Universal Robots PolyScope program: TEST_SUB_104RXFF.urp

Program TEST_SUB_104RXFF (installation=GD directory=/programs/GD createdIn=5.13.0 lastSavedIn=5.13.0 robotSerialNumber=20205000017)
Calibrated DH parameters: a=[-0.000157, -0.56303, -0.236706, -0.000074, -0.000109, 0]; d=[0.181705, 47.632387, 369.599619, -417.058513, 0.119878, 0.115667]; alpha=[1.570881, -0.005074, -0.001247, 1.56886, -1.570997, 0]; deltaTheta=[0, -0.405485, 5.544791, 1.143886, -0.000009, -0.000001]
InitVariablesNode
BeforeStart
  Script file /programs/GD/CONTROL/FORCE_CONTROL.script
    | def GET_TCP_FORCE_TOOL():
    |   force_torque=get_tcp_force()
    |   force_B=p[force_torque[0], force_torque[1], force_torque[2], 0, 0, 0]
    |   torque_B=p[force_torque[3], force_torque[4], force_torque[5], 0, 0, 0]
    |   tcp=get_actual_tcp_pose()
    |   rotation_BT=p[0, 0, 0, tcp[3], tcp[4], tcp[5]]
    |   force_T=pose_trans(pose_inv(rotation_BT), force_B)
    |   torque_T=pose_trans(pose_inv(rotation_BT), torque_B)
    |   force_torque_T=p[force_T[0], force_T[1], force_T[2], torque_T[0], torque_T[1], torque_T[2]]
    |   return force_torque_T
    | end
Robot Program (runOnlyOnce=true)
  SuppressedNode
    Script: SET_BUCKET()
  SuppressedNode
    Folder ROVI_CAPTURE
      If ( not ROVI_CAPTURE())
        SubPrgResult := rovi_err
        Wait Sleep waitTime=999999
      CandCnt := Y1[0]
      DistPillar := Y1[1] / 1000.0
      LevelZ := Y1[2] / 1000.0
      NeighborZ := Y1[3] / 1000.0
      If (GP_int_in[0]==1201)
        DistPillarBak := DistPillar
      If (CandCnt<1)
        SubPrgResult := 990
        Wait Sleep waitTime=999999
  SuppressedNode
    Folder ROVI_SOLVE
      If (CandCnt>0)
        Y2 := ROVI_SOLVE()
        If (Y2[0]≟10000.)
          SubPrgResult := rovi_err
          Wait Sleep waitTime=999999
  SuppressedNode
    UF := Y2
  DistPillar := 0.5
  Folder PICK
    SetPayload (workpieceName=k10)
    '1=MOVE'
    '2=MOVE+FIXEDBALANCE'
    '3=FORCEMOVE'
    '4=FORCEZ'
    '5=FORCEZ+WEAVE'
    '6=[LM]FORCEZ+WEAVE'
    '7=[RM]FORCEZ+WEAVE'
    '8=[RM]FORCEZ'
    i := 8
    Loop Counting (count=3) loopVariable(name=ループ_1)
      Switch expression=i
        Case (caseValue=1)
          MoveL speed 400 mm/s, acceleration 70 mm/s^2 (useActiveTCP=false) tcp=TCP_RX; feature=UF
            Waypoint Variable (Variable): variable(featureName=gGD_3_M_RX)
            Waypoint Variable (Variable): variable(featureName=gGD_2_M_RX)
            Wait Sleep waitTime=0.5
            SuppressedNode
              Popup Message (haltProgram=false message=ok? inputType=Text)
            Waypoint Variable (Variable): variable(featureName=gGD_1_M_RX)
        Case (caseValue=2)
          MoveL speed 400 mm/s, acceleration 70 mm/s^2 (useActiveTCP=false) tcp=TCP_RX; feature=UF
            Waypoint Variable (Variable): variable(featureName=gGD_3_M_RX)
            Waypoint Variable (Variable): variable(featureName=gGD_2_M_RX)
            Set SingleDigitalPulseActionState SingleDigitalPulseActionState(hiPulseInSeconds=1, pin=GP_bool_out[14])
            Wait Sleep waitTime=0.5
            SuppressedNode
              Popup Message (haltProgram=false message=ok? inputType=Text)
            Waypoint Variable (Variable): variable(featureName=gGD_1_M_RX)
            Set SingleDigitalPulseActionState SingleDigitalPulseActionState(hiPulseInSeconds=1, pin=GP_bool_out[15])
        Case (caseValue=3)
          MoveL speed 400 mm/s, acceleration 70 mm/s^2 (useActiveTCP=false) tcp=TCP_RX; feature=UF
            Waypoint Variable (Variable): variable(featureName=gGD_3_M_RX)
            Waypoint Variable (Variable): variable(featureName=gGD_2_M_RX)
            Set SingleDigitalPulseActionState SingleDigitalPulseActionState(hiPulseInSeconds=1, pin=GP_bool_out[14])
            Wait Sleep waitTime=0.5
            SuppressedNode
              Popup Message (haltProgram=false message=ok? inputType=Text)
          Force Frame feature=Joint_6_name; selection=[1, 1, 0, 0, 0, 0]; wrench=[0, 0, 0, 0, 0, 0]; limitsForce=[0.005, 0.005, 0.03, 1.047198, 1.047198, 1.047198]; limitsMotion=[0.1, 0.1, 0.1, 0.349066, 0.349066, 0.349066]
            MoveL speed 120 mm/s, acceleration 70 mm/s^2 (useActiveTCP=false) tcp=TCP_RX; feature=UF
              Waypoint Variable (Variable): variable(featureName=gGD_1_M_RX)
          Set SingleDigitalPulseActionState SingleDigitalPulseActionState(hiPulseInSeconds=1, pin=GP_bool_out[15])
        Case (caseValue=4)
          MoveL speed 400 mm/s, acceleration 70 mm/s^2 (useActiveTCP=false) tcp=TCP_RX; feature=UF
            Waypoint Variable (Variable): variable(featureName=gGD_3_M_RX)
            Waypoint Variable (Variable): variable(featureName=gGD_2_M_RX)
            Set SingleDigitalPulseActionState SingleDigitalPulseActionState(hiPulseInSeconds=1, pin=GP_bool_out[14])
            Wait Sleep waitTime=0.5
            SuppressedNode
              Popup Message (haltProgram=false message=ok? inputType=Text)
          Force Frame feature=Joint_6_name; selection=[1, 1, 1, 0, 0, 0]; wrench=[0, 0, 10, 0, 0, 0]; limitsForce=[0.005, 0.005, 0.03, 0.034907, 0.034907, 1.047198]; limitsMotion=[0.1, 0.1, 0.1, 0.349066, 0.349066, 0.349066]
            Wait Condition expression=CurrPos_p[1]≤(gGD_1_M_RX[1]-0.015)
          Popup Message (haltProgram=false message=ok inputType=Text)
          Set SingleDigitalPulseActionState SingleDigitalPulseActionState(hiPulseInSeconds=1, pin=GP_bool_out[15])
        Case (caseValue=5)
          MoveL speed 400 mm/s, acceleration 70 mm/s^2 (useActiveTCP=false) tcp=TCP_RX; feature=UF
            Waypoint Variable (Variable): variable(featureName=gGD_3_M_RX)
            Waypoint Variable (Variable): variable(featureName=gGD_2_M_RX)
            Set SingleDigitalPulseActionState SingleDigitalPulseActionState(hiPulseInSeconds=1, pin=GP_bool_out[14])
            Wait Sleep waitTime=0.5
            SuppressedNode
              Popup Message (haltProgram=false message=ok? inputType=Text)
          Sub3100_Option := 9
          Force Frame feature=Joint_6_name; selection=[1, 1, 1, 0, 0, 0]; wrench=[0, 0, 10, 0, 0, 0]; limitsForce=[0.005, 0.005, 0.03, 0.034907, 0.034907, 1.047198]; limitsMotion=[0.1, 0.1, 0.1, 0.349066, 0.349066, 0.349066]
            Loop While (checkContinuously=false) expression=CurrPos_p[1]>(gGD_1_M_RX[1]-0.015)
              If tcp_speed[2]<0.0005
                '7:RX+,8:RX-,9:RY+,10:RY-,11:RZ+,12:RZ-'
                Sub3100_Xd := [0.,0.,0.,0.,0.,0.]
                Sub3100_q := floor((Sub3100_Option-1) / 2)
                Sub3100_e := 1-((Sub3100_Option-1) % 2)*2
                Sub3100_t := 0.2
                Script: Sub3100_Xd[Sub3100_q]=d2r(Sub3100_XdRot)*Sub3100_e
                Script: speedl(Sub3100_Xd,Sub3100_aRot,Sub3100_t)
                If Sub3100_Option≟9
                  Sub3100_Option := 10
                Else 
                  Sub3100_Option := 9
          Popup Message (haltProgram=false message=ok inputType=Text)
          Set SingleDigitalPulseActionState SingleDigitalPulseActionState(hiPulseInSeconds=1, pin=GP_bool_out[15])
        Case (caseValue=6)
          MoveL speed 400 mm/s, acceleration 70 mm/s^2 (useActiveTCP=false) tcp=TCP_RX; feature=UF
            Waypoint Variable (Variable): variable(featureName=gGD_3_LM_RX)
            Waypoint Variable (Variable): variable(featureName=gGD_2_LM_RX)
            Set SingleDigitalPulseActionState SingleDigitalPulseActionState(hiPulseInSeconds=1, pin=GP_bool_out[14])
            Wait Sleep waitTime=0.5
            SuppressedNode
              Popup Message (haltProgram=false message=ok? inputType=Text)
          Sub3100_Option := 9
          Force Frame feature=Joint_6_name; selection=[1, 1, 1, 0, 0, 0]; wrench=[0, 0, 10, 0, 0, 0]; limitsForce=[0.005, 0.005, 0.03, 0.034907, 0.034907, 1.047198]; limitsMotion=[0.1, 0.1, 0.1, 0.349066, 0.349066, 0.349066]
            Loop While (checkContinuously=false) expression=CurrPos_p[1]>(gGD_1_LM_RX[1]-0.015)
              If tcp_speed[2]<0.0005
                '7:RX+,8:RX-,9:RY+,10:RY-,11:RZ+,12:RZ-'
                Sub3100_Xd := [0.,0.,0.,0.,0.,0.]
                Sub3100_q := floor((Sub3100_Option-1) / 2)
                Sub3100_e := 1-((Sub3100_Option-1) % 2)*2
                Sub3100_t := 0.2
                Script: Sub3100_Xd[Sub3100_q]=d2r(Sub3100_XdRot)*Sub3100_e
                Script: speedl(Sub3100_Xd,Sub3100_aRot/2.0,Sub3100_t)
                If Sub3100_Option≟9
                  Sub3100_Option := 10
                Else 
                  Sub3100_Option := 9
          Popup Message (haltProgram=false message=ok inputType=Text)
          Set SingleDigitalPulseActionState SingleDigitalPulseActionState(hiPulseInSeconds=1, pin=GP_bool_out[15])
        Case (caseValue=7)
          MoveL speed 400 mm/s, acceleration 70 mm/s^2 (useActiveTCP=false) tcp=TCP_RX; feature=UF
            Waypoint Variable (Variable): variable(featureName=gGD_3_RM_RX)
            Waypoint Variable (Variable): variable(featureName=gGD_2_RM_RX)
            Set SingleDigitalPulseActionState SingleDigitalPulseActionState(hiPulseInSeconds=1, pin=GP_bool_out[14])
            Wait Sleep waitTime=0.5
            SuppressedNode
              Popup Message (haltProgram=false message=ok? inputType=Text)
          Sub3100_Option := 9
          Force Frame feature=Joint_6_name; selection=[1, 1, 1, 0, 0, 0]; wrench=[0, 0, 10, 0, 0, 0]; limitsForce=[0.005, 0.005, 0.03, 0.034907, 0.034907, 1.047198]; limitsMotion=[0.1, 0.1, 0.1, 0.349066, 0.349066, 0.349066]
            Loop While (checkContinuously=false) expression=CurrPos_p[1]>(gGD_1_RM_RX[1]-0.015)
              If tcp_speed[2]<0.0005
                '7:RX+,8:RX-,9:RY+,10:RY-,11:RZ+,12:RZ-'
                Sub3100_Xd := [0.,0.,0.,0.,0.,0.]
                Sub3100_q := floor((Sub3100_Option-1) / 2)
                Sub3100_e := 1-((Sub3100_Option-1) % 2)*2
                Sub3100_t := 0.2
                Script: Sub3100_Xd[Sub3100_q]=d2r(Sub3100_XdRot)*Sub3100_e
                Script: speedl(Sub3100_Xd,Sub3100_aRot/2.0,Sub3100_t)
                If Sub3100_Option≟9
                  Sub3100_Option := 10
                Else 
                  Sub3100_Option := 9
          Popup Message (haltProgram=false message=ok inputType=Text)
          Set SingleDigitalPulseActionState SingleDigitalPulseActionState(hiPulseInSeconds=1, pin=GP_bool_out[15])
        Case (caseValue=8)
          MoveL speed 400 mm/s, acceleration 70 mm/s^2 (useActiveTCP=false) tcp=TCP_RX; feature=UF
            Waypoint Variable (Variable): variable(featureName=gGD_3_RM_RX)
            Waypoint Variable (Variable): variable(featureName=gGD_2_RM_RX)
            Set SingleDigitalPulseActionState SingleDigitalPulseActionState(hiPulseInSeconds=1, pin=GP_bool_out[14])
            Wait Sleep waitTime=0.5
            SuppressedNode
              Popup Message (haltProgram=false message=ok? inputType=Text)
          Force Frame feature=Joint_6_name; selection=[1, 1, 1, 0, 0, 0]; wrench=[0, 0, 10, 0, 0, 0]; limitsForce=[0.005, 0.005, 0.03, 0.034907, 0.034907, 1.047198]; limitsMotion=[0.1, 0.1, 0.1, 0.349066, 0.349066, 0.349066]
            Wait Condition expression=CurrPos_p[1]≤(gGD_1_RM_RX[1]-0.015)
          Popup Message (haltProgram=false message=ok inputType=Text)
          Set SingleDigitalPulseActionState SingleDigitalPulseActionState(hiPulseInSeconds=1, pin=GP_bool_out[15])
      If i<6
        MoveL speed 400 mm/s, acceleration 70 mm/s^2 (useActiveTCP=false) tcp=TCP_RX; feature=UF
          Waypoint Variable (Variable): variable(featureName=gGD_2_M_RX)
          Waypoint Variable (Variable): variable(featureName=gGD_3_M_RX)
      ElseIf i≟6
        MoveL speed 400 mm/s, acceleration 70 mm/s^2 (useActiveTCP=false) tcp=TCP_RX; feature=UF
          Waypoint Variable (Variable): variable(featureName=gGD_2_LM_RX)
          Waypoint Variable (Variable): variable(featureName=gGD_3_LM_RX)
      Else 
        MoveL speed 400 mm/s, acceleration 70 mm/s^2 (useActiveTCP=false) tcp=TCP_RX; feature=UF
          Waypoint Variable (Variable): variable(featureName=gGD_2_RM_RX)
          Waypoint Variable (Variable): variable(featureName=gGD_3_RM_RX)
      Wait Sleep waitTime=4
    Halt
    If (0≤DistPillar and DistPillar≤DistPillarAPTh)
      MoveL speed 400 mm/s, acceleration 140 mm/s^2 (useActiveTCP=false) tcp=TCP_1; feature=UF
        Waypoint Variable (Variable): variable(featureName=gGD_4_LM)
      MoveL speed 400 mm/s, acceleration 140 mm/s^2 (useActiveTCP=false) tcp=TCP_RX; feature=UF
        Waypoint Variable (Variable): variable(featureName=gGD_3_LM_RX)
        Waypoint Variable (Variable): variable(featureName=gGD_2_LM_RX)
        Set SingleDigitalPulseActionState SingleDigitalPulseActionState(hiPulseInSeconds=1, pin=GP_bool_out[14])
        Wait Sleep waitTime=0.5
        SuppressedNode
          Popup Message (haltProgram=false message=ok? inputType=Text)
        Waypoint Variable (Variable): variable(featureName=gGD_1_LM_RX)
      Sub3100_Option := 9
      Force Frame feature=Joint_6_name; selection=[1, 1, 1, 0, 0, 0]; wrench=[0, 0, 10, 0, 0, 0]; limitsForce=[0.005, 0.005, 0.03, 0.034907, 0.034907, 1.047198]; limitsMotion=[0.1, 0.1, 0.1, 0.349066, 0.349066, 0.349066]
        Loop While (checkContinuously=false) expression=CurrPos_p[1]>(gGD_1_M_RX[1]-0.015)
          If tcp_speed[2]<0.0005
            '7:RX+,8:RX-,9:RY+,10:RY-,11:RZ+,12:RZ-'
            Sub3100_Xd := [0.,0.,0.,0.,0.,0.]
            Sub3100_q := floor((Sub3100_Option-1) / 2)
            Sub3100_e := 1-((Sub3100_Option-1) % 2)*2
            Sub3100_t := 0.2
            Script: Sub3100_Xd[Sub3100_q]=d2r(Sub3100_XdRot)*Sub3100_e
            Script: speedl(Sub3100_Xd,Sub3100_aRot,Sub3100_t)
            If Sub3100_Option≟9
              Sub3100_Option := 10
            Else 
              Sub3100_Option := 9
      Set SingleDigitalPulseActionState SingleDigitalPulseActionState(hiPulseInSeconds=1, pin=GP_bool_out[15])
    ElseIf (-DistPillarAPTh≤DistPillar and DistPillar≤0)
      MoveL speed 400 mm/s, acceleration 70 mm/s^2 (useActiveTCP=false) tcp=TCP_1; feature=UF
        Waypoint Variable (Variable): variable(featureName=gGD_4_RM)
      MoveL speed 400 mm/s, acceleration 70 mm/s^2 (useActiveTCP=false) tcp=TCP_RX; feature=UF
        Waypoint Variable (Variable): variable(featureName=gGD_3_RM_RX)
        Waypoint Variable (Variable): variable(featureName=gGD_2_RM_RX)
        Wait Sleep waitTime=0.5
        SuppressedNode
          Popup Message (haltProgram=false message=ok? inputType=Text)
        Waypoint Variable (Variable): variable(featureName=gGD_1_RM_RX)
    Else 
      MoveL speed 400 mm/s, acceleration 70 mm/s^2 (useActiveTCP=false) tcp=TCP_RX; feature=UF
        Waypoint Variable (Variable): variable(featureName=gGD_3_M_RX)
        Waypoint Variable (Variable): variable(featureName=gGD_2_M_RX)
        Set SingleDigitalPulseActionState SingleDigitalPulseActionState(hiPulseInSeconds=1, pin=GP_bool_out[14])
        Wait Sleep waitTime=0.5
        SuppressedNode
          Popup Message (haltProgram=false message=ok? inputType=Text)
      Force Frame feature=Joint_6_name; selection=[1, 1, 0, 0, 0, 0]; wrench=[0, 0, 0, 0, 0, 0]; limitsForce=[0.005, 0.005, 0.03, 1.047198, 1.047198, 1.047198]; limitsMotion=[0.1, 0.1, 0.1, 0.349066, 0.349066, 0.349066]
        MoveL speed 120 mm/s, acceleration 70 mm/s^2 (useActiveTCP=false) tcp=TCP_RX; feature=UF
          Waypoint Variable (Variable): variable(featureName=gGD_1_M_RX)
      Set SingleDigitalPulseActionState SingleDigitalPulseActionState(hiPulseInSeconds=1, pin=GP_bool_out[15])
      Wait Sleep waitTime=2
      Popup Message (haltProgram=false message=force done! inputType=Text)
    If ( not GPBI_WorkExists)
      SubPrgResult := 821
      Wait Sleep waitTime=999999
Thread スレッド_1 (runOnlyOnce=false)
  Script: CurrPos_p=get_actual_tcp_pose()
  tcp_speed := get_actual_tcp_speed()
  tcp_force_tool := GET_TCP_FORCE_TOOL()
  Script: sync()
